TYPE ST_InstFeedback :
STRUCT
	ChargerVolt : REAL;
	CapVolt		: ARRAY [1..15] OF REAL;
	Cur  		: REAL;
	TotalVoltage: REAL;
END_STRUCT
END_TYPE

(* stored: Version 1.1.0.1, ProductVersion 3.1.4024.11
   DUT ST_InstFeedback: Id {b18a5ab0-4514-44df-a73d-05cbf568e132} *)
